{library PUBLIC}
(*
 Function type, to be used in DataGram structure to specify set of functions.

 Note that values <=0 are return values only.
 *)
TYPE FUNCTION_TYPE : 
(
	FUNCTION_TYPE_ERROR_BUSY:=-2,				(* Old function call is not ready  *)
	FUNCTION_TYPE_ERROR_NO_FUNCTION:=-1,		(* RPC function not found *)
	FUNCTION_TYPE_TASK_STARTED:=0,				(* ASynchronous function started *)
	FUNCTION_TYPE_ASYNC_RPC:=1,					(* ASynchronous RPC *)
	FUNCTION_TYPE_SYNC_RPC,   					(* Synchronous RPC *)
	FUNCTION_TYPE_INFORMATION					(* Synchronous RPC dedicated for status functions *)
);
END_TYPE
//  FUNCTION_TYPE_ERROR_BUSY = '-2'
//  FUNCTION_TYPE_ERROR_NO_FUNCTION = '-1'

(* stored: Version 1.1.0.1, ProductVersion 3.1.4024.2
   EnumerationTextList FUNCTION_TYPE: Id {629425d9-b638-4180-9b59-d3c6cc4e15d7} *)
